FUNCTION_BLOCK FB_SV_Ablaufsteuerung
VAR_IN_OUT
	Zustand			: ST_SV_Zustand;
	Stellwert		: ST_SV_Stellwert;
END_VAR
VAR_INPUT
	Steuerung		: ST_SV_Steuerung;
	Parameter		: ST_SV_Parameter;
END_VAR
VAR_OUTPUT
END_VAR
VAR
	Timer		: TON;
END_VAR

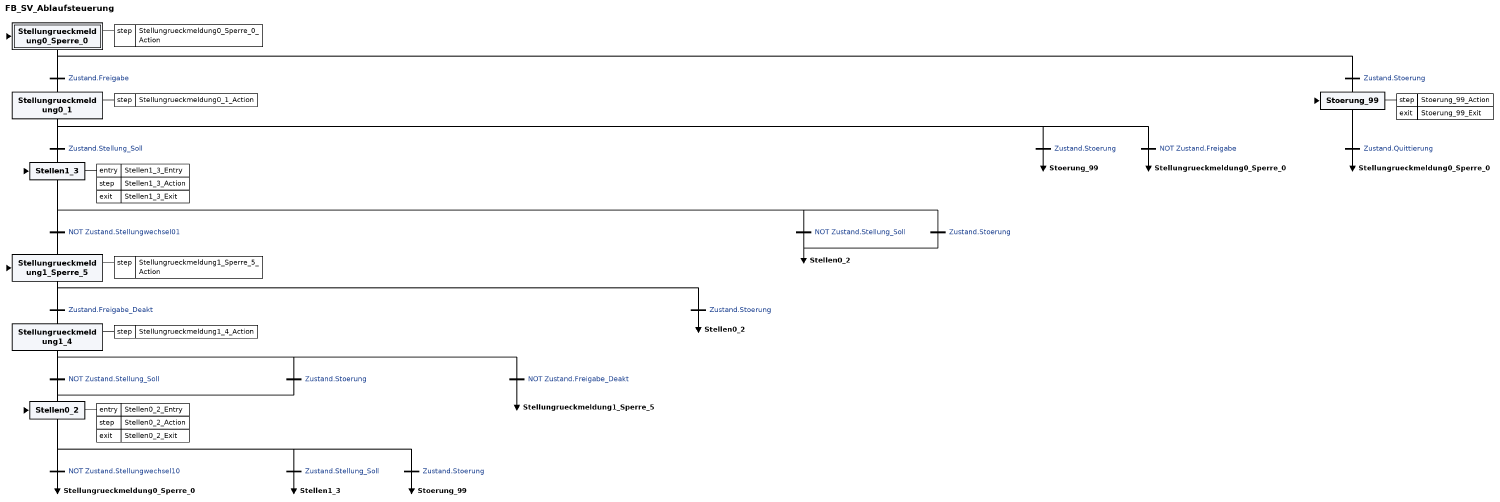
INITIAL_STEP Stellungrueckmeldung0_Sperre_0:
    Stellungrueckmeldung0_Sperre_0_Action(N);  // step action
END_STEP
TRANSITION FROM Stellungrueckmeldung0_Sperre_0 TO Stellungrueckmeldung0_1
    := Zustand.Freigabe;
END_TRANSITION
TRANSITION FROM Stellungrueckmeldung0_Sperre_0 TO Stoerung_99
    := Zustand.Stoerung;
END_TRANSITION
STEP Stoerung_99:
    Stoerung_99_Action(N);  // step action
    Stoerung_99_Exit(P0);  // exit action
END_STEP
TRANSITION FROM Stoerung_99 TO Stellungrueckmeldung0_Sperre_0
    := Zustand.Quittierung;
END_TRANSITION
STEP Stellungrueckmeldung0_1:
    Stellungrueckmeldung0_1_Action(N);  // step action
END_STEP
TRANSITION FROM Stellungrueckmeldung0_1 TO Stellen1_3
    := Zustand.Stellung_Soll;
END_TRANSITION
TRANSITION FROM Stellungrueckmeldung0_1 TO Stoerung_99
    := Zustand.Stoerung;
END_TRANSITION
TRANSITION FROM Stellungrueckmeldung0_1 TO Stellungrueckmeldung0_Sperre_0
    := NOT Zustand.Freigabe;
END_TRANSITION
STEP Stellen1_3:
    Stellen1_3_Entry(P1);  // entry action
    Stellen1_3_Action(N);  // step action
    Stellen1_3_Exit(P0);  // exit action
END_STEP
TRANSITION FROM Stellen1_3 TO Stellungrueckmeldung1_Sperre_5
    := NOT Zustand.Stellungwechsel01;
END_TRANSITION
TRANSITION FROM Stellen1_3 TO Stellen0_2
    := NOT Zustand.Stellung_Soll;
END_TRANSITION
TRANSITION FROM Stellen1_3 TO Stellen0_2
    := Zustand.Stoerung;
END_TRANSITION
STEP Stellungrueckmeldung1_Sperre_5:
    Stellungrueckmeldung1_Sperre_5_Action(N);  // step action
END_STEP
TRANSITION FROM Stellungrueckmeldung1_Sperre_5 TO Stellungrueckmeldung1_4
    := Zustand.Freigabe_Deakt;
END_TRANSITION
TRANSITION FROM Stellungrueckmeldung1_Sperre_5 TO Stellen0_2
    := Zustand.Stoerung;
END_TRANSITION
STEP Stellungrueckmeldung1_4:
    Stellungrueckmeldung1_4_Action(N);  // step action
END_STEP
TRANSITION FROM Stellungrueckmeldung1_4 TO Stellen0_2
    := NOT Zustand.Stellung_Soll;
END_TRANSITION
TRANSITION FROM Stellungrueckmeldung1_4 TO Stellen0_2
    := Zustand.Stoerung;
END_TRANSITION
TRANSITION FROM Stellungrueckmeldung1_4 TO Stellungrueckmeldung1_Sperre_5
    := NOT Zustand.Freigabe_Deakt;
END_TRANSITION
STEP Stellen0_2:
    Stellen0_2_Entry(P1);  // entry action
    Stellen0_2_Action(N);  // step action
    Stellen0_2_Exit(P0);  // exit action
END_STEP
TRANSITION FROM Stellen0_2 TO Stellungrueckmeldung0_Sperre_0
    := NOT Zustand.Stellungwechsel10;
END_TRANSITION
TRANSITION FROM Stellen0_2 TO Stellen1_3
    := Zustand.Stellung_Soll;
END_TRANSITION
TRANSITION FROM Stellen0_2 TO Stoerung_99
    := Zustand.Stoerung;
END_TRANSITION

ACTION Stellen0_2_Action:
(* Nachlauf Timer starten *)
Timer( 	IN := Zustand.Stellungwechsel10,
		PT := DINT_TO_TIME(Parameter.Zeit_Stellen0),
);
Zustand.Stellungwechsel10	:= NOT Timer.Q;

(* Stellwert setzen *)
Stellwert.Stellung := FALSE;

(* Zustand setzen *)
Zustand.Status := E_Stellventil_Zustand_Stellungwechsel10;
END_ACTION

ACTION Stellen0_2_Entry:
(* Reset Timer *)
Timer(IN := FALSE);
Zustand.Stellungwechsel10 := TRUE;
END_ACTION

ACTION Stellen0_2_Exit:
Zustand.Stellungwechsel10 := FALSE;
END_ACTION

ACTION Stellen1_3_Action:
(* Vorlaufzeit Timer starten *)
Timer( 	IN := Zustand.Stellungwechsel01,
		PT := DINT_TO_TIME(Parameter.Zeit_Stellen1),
);
Zustand.Stellungwechsel01	:= NOT Timer.Q;

(* Stellwert setzen *)
Stellwert.Stellung := TRUE;

(* Zustand setzen *)
Zustand.Status := E_Stellventil_Zustand_Stellungwechsel01;
END_ACTION

ACTION Stellen1_3_Entry:
(* Reset Timer *)
Timer(IN := FALSE);
Zustand.Stellungwechsel01 := TRUE;
END_ACTION

ACTION Stellen1_3_Exit:
Zustand.Stellungwechsel01 := FALSE;
END_ACTION

ACTION Stellungrueckmeldung0_1_Action:
(* Stellwert setzen *)
Stellwert.Stellung := FALSE;
Zustand.Stellung := FALSE;

(* Zustand setzen *)
Zustand.Status := E_Stellventil_Zustand_Status_Stellungrueckmeldung0;
END_ACTION

ACTION Stellungrueckmeldung0_Sperre_0_Action:
(* Stellwert setzen *)
Stellwert.Stellung := FALSE;
Zustand.Stellung := FALSE;

(* Zustand setzen *)
Zustand.Status := E_Stellventil_Zustand_Status_Stellungrueckmeldung0_Sperre;
END_ACTION

ACTION Stellungrueckmeldung1_4_Action:
(* Stellwert setzen *)
Stellwert.Stellung := TRUE;
Zustand.Stellung := TRUE;

(* Zustand setzen *)
Zustand.Status := E_Stellventil_Zustand_Status_Stellungrueckmeldung1;
END_ACTION

ACTION Stellungrueckmeldung1_Sperre_5_Action:
(* Stellwert setzen *)
Stellwert.Stellung := TRUE;
Zustand.Stellung := TRUE;

(* Zustand setzen *)
Zustand.Status := E_Stellventil_Zustand_Status_Stellungrueckmeldung1_Sperre;
END_ACTION

ACTION Stoerung_99_Action:
(* Stellwert setzen *)
Stellwert.Stellung := Zustand.Stellung;

(* Zustand setzen *)
Zustand.Stoerung := TRUE;
Zustand.Status := E_PU_Zustand_Status_Stoerung;
END_ACTION

ACTION Stoerung_99_Exit:
Zustand.Stoerung	:= FALSE;
END_ACTION

END_FUNCTION_BLOCK

(* stored: Version 1.1.0.1, ProductVersion 3.1.4024.9
   POU FB_SV_Ablaufsteuerung: Id {d42aba02-f65f-4f07-a5b0-1b76b7a7eb7e}, SpecialFunc None
   Action Stellen0_2_Action: Id {40309867-551d-45ee-8176-ca175fc9b178}
   Action Stellen0_2_Entry: Id {7343d578-6408-4139-8b4c-1ecedac27a4a}
   Action Stellen0_2_Exit: Id {b66fd9db-8e28-44dd-a84c-f98ec2c584fc}
   Action Stellen1_3_Action: Id {ff58e86d-c3fd-4603-9d93-92253bd2e7f8}
   Action Stellen1_3_Entry: Id {e54eb886-fd3c-43b7-8e58-ed18199c5a83}
   Action Stellen1_3_Exit: Id {09a4789a-3dd4-4bb5-bf0e-68f7011e912c}
   Action Stellungrueckmeldung0_1_Action: Id {b638ecde-beb9-4889-9d37-e2d34f97bbb3}
   Action Stellungrueckmeldung0_Sperre_0_Action: Id {97609f2f-ecdd-4231-ac6c-146bf77fcc91}
   Action Stellungrueckmeldung1_4_Action: Id {fb9decaf-c1c0-4eea-9d1c-c22858e74868}
   Action Stellungrueckmeldung1_Sperre_5_Action: Id {dbd62c8d-3bfe-4678-91e1-a1358f8eb3ea}
   Action Stoerung_99_Action: Id {beb7cb51-e6b3-4555-b704-511c8d93ae82}
   Action Stoerung_99_Exit: Id {b03610cc-469c-4519-a26a-cd4e5407f529} *)
